INTERFACE I_QueryInterface EXTENDS __SYSTEM.IQueryInterface

END_INTERFACE

(* stored: Version 1.1.0.1, ProductVersion 3.1.4024.4
   Itf I_QueryInterface: Id {08c3cc90-4bba-0ae2-3db8-665a0b556a60} *)
